TYPE "udt_MbClient"
VERSION : 0.1
// Block: udt_MbClient
   STRUCT
      req : Bool;
      disconnect : Bool;
      mode : USInt;
      DataAddr : UDInt;
      DataLen : UInt;
      connect : TCON_IP_v4;
   END_STRUCT;

END_TYPE
